FUNCTION_BLOCK FB_inRange
VAR_INPUT
	in_istPos 	:REAL;
	in_sollPos	:REAL;
	in_Fenster	:REAL;
END_VAR
VAR_OUTPUT
	out_imBereich :BOOL;
END_VAR
VAR
END_VAR

 out_imBereich := 	in_istPos > in_sollPos - in_Fenster
 					AND in_istPos < in_sollPos + in_Fenster;

END_FUNCTION_BLOCK

(* stored: Version 1.1.0.1
   POU FB_inRange: Id {001d83f7-815e-488e-ae0d-8a20c0131bc6}, SpecialFunc None *)
